// TIA Portal V17 export
// export: Created 2026-04-13T11:12:43.7188239Z, ExportSetting WithDefaults, DisplayName Totally Integrated Automation Portal, DisplayVersion V17 Update 4, DisplayName TIA Portal Openness, DisplayVersion V17 Update 4, DisplayName TIA Portal Version Control Interface, DisplayVersion V17, DisplayName SINAMICS Startdrive Advanced, DisplayVersion V17, DisplayName SINAMICS Startdrive G130, G150, S120, S150, SINAMICS MV, S210, DisplayVersion V17, DisplayName SINAMICS Startdrive G110M, G120, G120C, G120D, G120P, G115D, DisplayVersion V17, DisplayName STEP 7 Professional, DisplayVersion V17 Update 4, DisplayName STEP 7 Safety, DisplayVersion V17, DisplayName WinCC Professional, DisplayVersion V17 Update 4
FUNCTION_BLOCK "32-油炉控制"   // FB22, LAD
{ S7_Optimized_Access := 'FALSE' }
VERSION : 0.1
// stored: AutoNumber true, IsIECCheckEnabled false, SetENOAutomatically false, UDAEnableTagReadback false
   VAR_IN_OUT
      油炉温度写 : Real;
      油炉温度读 : Real;
      油炉循环泵启停 : Bool;
      油炉报警 : Bool;
      油炉冷却阀启停状态 : Bool;
      油炉加热泵启停状态 : Bool;
      油炉加热器1状态 : Bool;
      油炉加热器2状态 : Bool;
      油炉运行状态 : Bool;
      油炉自整定状态 : Bool;
      油炉强制冷却状态 : Bool;
      YL油炉温度写读 : Real;
   END_VAR
   VAR
      MB_COMM_LOAD { S7_SetPoint := 'True'} : Modbus_Comm_Load;
      MB_MASTER_DB { S7_SetPoint := 'True'} : Modbus_Master;
   END_VAR
   VAR DB_SPECIFIC
      CTU { S7_SetPoint := 'True'} : CTU_INT;
      TEMP { S7_SetPoint := 'True'} : Bool;
      TP : Array[0..40] of Bool;
      油炉温度读辅 : Int;
      油炉温度写辅 : Int;
      ST1 : Real;
      ST2 : Real;
      ST3 : Real;
      ST4 : Real;
      ST5 : Real;
      ST16 : Real;
      ST17 : Real;
      ST18 : Real;
      ST20 : Real;
      ST21 : Real;
      ST22 : Real;
      油炉状态1 : Int;
      油炉状态2 : Int;
      油炉启停字 : Int;
      油炉加热状态 : Int;
      油炉运行标志 : Int;
      YL油炉温度写读辅 : Int;
   END_VAR
   VAR
      Modbus_Comm_Load { S7_SetPoint := 'True'} : Modbus_Comm_Load;
      Modbus_Master { S7_SetPoint := 'True'} : Modbus_Master;
   END_VAR
   VAR_TEMP   // added for the SCL form of the ladder/FBD networks
      _w1 : Bool;
      _w2 : Bool;
      _w3 : Bool;
   END_VAR
BEGIN

REGION Network 1
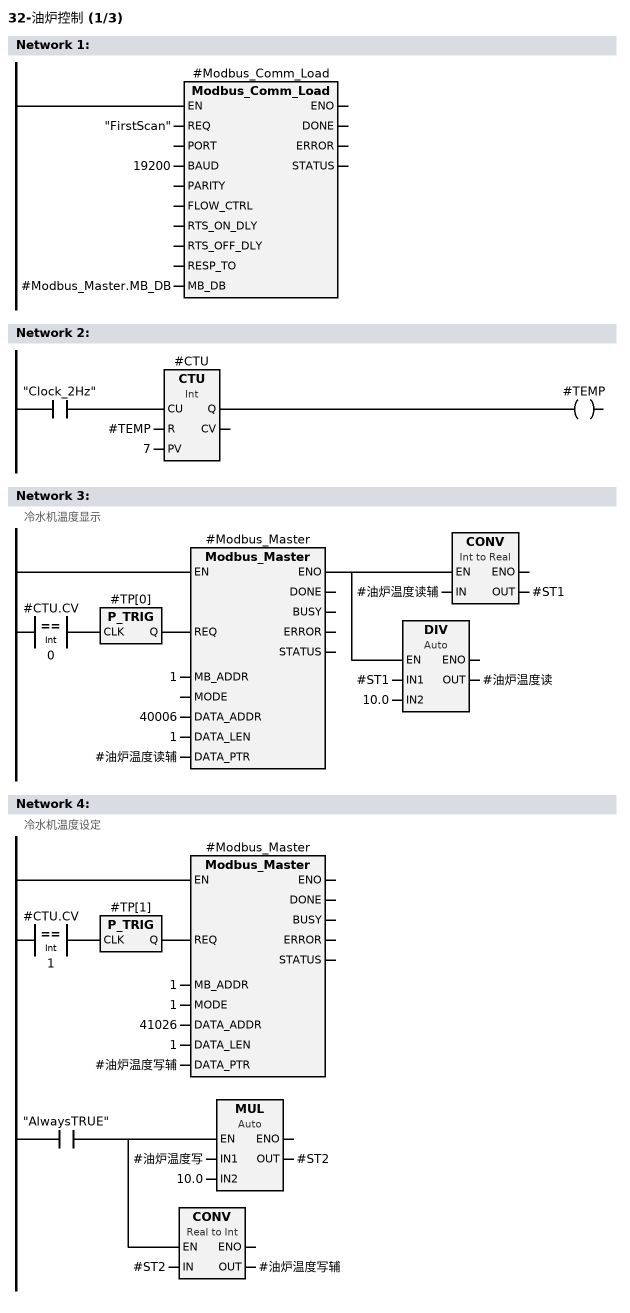
   RUNG wire#powerrail
      #Modbus_Comm_Load.Modbus_Comm_Load(REQ := "FirstScan", PORT :=, BAUD := 19200, PARITY :=, FLOW_CTRL :=, RTS_ON_DLY :=, RTS_OFF_DLY :=, RESP_TO :=, MB_DB := #Modbus_Master.MB_DB, DONE =>, ERROR =>, STATUS =>)
   END_RUNG
   // the same network as SCL:
   #Modbus_Comm_Load(REQ := "FirstScan", BAUD := 19200, MB_DB := #Modbus_Master.MB_DB);   // Modbus_Comm_Load
END_REGION

REGION Network 2
   RUNG wire#powerrail
      Contact( "Clock_2Hz" )
      { S7_Templates := "value_type := Int" } #CTU.CTU(r := #TEMP, pv := 7, cv =>)
      Coil( #TEMP )
   END_RUNG
   // the same network as SCL:
   #CTU(CU := "Clock_2Hz", R := #TEMP, PV := 7);   // CTU
   #TEMP := #CTU.Q;
END_REGION

REGION Network 3
   // 冷水机温度显示
   RUNG wire#powerrail
      #Modbus_Master.Modbus_Master(REQ := wire#w1, MB_ADDR := 1, MODE :=, DATA_ADDR := 40006, DATA_LEN := 1, DATA_PTR := #油炉温度读辅, DONE =>, BUSY =>, ERROR =>, STATUS =>)
      wire#w2
      { S7_Templates := "[SrcType := Int, DestType := Real]" } Convert(in := #油炉温度读辅, out => #ST1)
   END_RUNG
   RUNG wire#powerrail
      { S7_Templates := "SrcType := Int" } EQ_Contact(in1 := #CTU.CV, in2 := 0)
      P_Trig( #TP[0] )
   END_RUNG wire#w1
   RUNG wire#w2
      Div(in1 := #ST1, in2 := 10.0, out => #油炉温度读)
   END_RUNG
   // the same network as SCL:
   #_w1 := #CTU.CV = 0;
   #_w2 := #_w1 AND NOT #TP[0];   // rising edge
   #TP[0] := #_w1;
   #Modbus_Master(REQ := #_w2,   // Modbus_Master
                  MB_ADDR := 1,
                  DATA_ADDR := 40006,
                  DATA_LEN := 1,
                  DATA_PTR := #油炉温度读辅,
                  ENO => #_w3);
   IF #_w3 THEN
       #ST1 := INT_TO_REAL(#油炉温度读辅);
       #油炉温度读 := #ST1 / 10.0;
   END_IF;
END_REGION

REGION Network 4
   // 冷水机温度设定
   RUNG wire#powerrail
      #Modbus_Master.Modbus_Master(REQ := wire#w1, MB_ADDR := 1, MODE := 1, DATA_ADDR := 41026, DATA_LEN := 1, DATA_PTR := #油炉温度写辅, DONE =>, BUSY =>, ERROR =>, STATUS =>)
   END_RUNG
   RUNG wire#powerrail
      { S7_Templates := "SrcType := Int" } EQ_Contact(in1 := #CTU.CV, in2 := 1)
      P_Trig( #TP[1] )
   END_RUNG wire#w1
   RUNG wire#powerrail
      Contact( "AlwaysTRUE" )
      wire#w2
      Mul(in1 := #油炉温度写, in2 := 10.0, out => #ST2)
   END_RUNG
   RUNG wire#w2
      { S7_Templates := "[SrcType := Real, DestType := Int]" } Convert(in := #ST2, out => #油炉温度写辅)
   END_RUNG
   // the same network as SCL:
   #_w1 := #CTU.CV = 1;
   #_w2 := #_w1 AND NOT #TP[1];   // rising edge
   #TP[1] := #_w1;
   #Modbus_Master(REQ := #_w2, MB_ADDR := 1, MODE := 1, DATA_ADDR := 41026, DATA_LEN := 1, DATA_PTR := #油炉温度写辅);   // Modbus_Master
   IF "AlwaysTRUE" THEN
       #ST2 := #油炉温度写 * 10.0;
       #油炉温度写辅 := REAL_TO_INT(#ST2);
   END_IF;
END_REGION

REGION Network 5
   // 冷水机温度设定
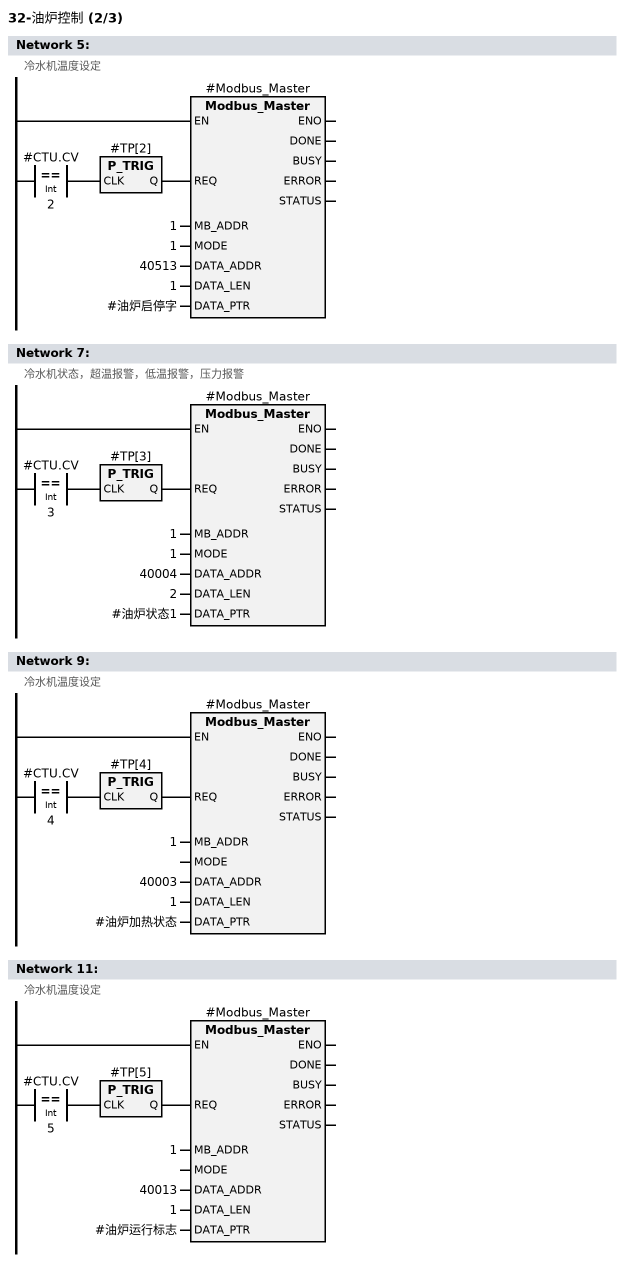
   RUNG wire#powerrail
      #Modbus_Master.Modbus_Master(REQ := wire#w1, MB_ADDR := 1, MODE := 1, DATA_ADDR := 40513, DATA_LEN := 1, DATA_PTR := #油炉启停字, DONE =>, BUSY =>, ERROR =>, STATUS =>)
   END_RUNG
   RUNG wire#powerrail
      { S7_Templates := "SrcType := Int" } EQ_Contact(in1 := #CTU.CV, in2 := 2)
      P_Trig( #TP[2] )
   END_RUNG wire#w1
   // the same network as SCL:
   #_w1 := #CTU.CV = 2;
   #_w2 := #_w1 AND NOT #TP[2];   // rising edge
   #TP[2] := #_w1;
   #Modbus_Master(REQ := #_w2, MB_ADDR := 1, MODE := 1, DATA_ADDR := 40513, DATA_LEN := 1, DATA_PTR := #油炉启停字);   // Modbus_Master
END_REGION

REGION Network 6 (SCL)
   IF #油炉循环泵启停 = TRUE THEN
       #油炉启停字:= 114;
   ELSE
       #油炉启停字 := 112;
   END_IF;
END_REGION

REGION Network 7
   // 冷水机状态，超温报警，低温报警，压力报警
   RUNG wire#powerrail
      #Modbus_Master.Modbus_Master(REQ := wire#w1, MB_ADDR := 1, MODE := 1, DATA_ADDR := 40004, DATA_LEN := 2, DATA_PTR := #油炉状态1, DONE =>, BUSY =>, ERROR =>, STATUS =>)
   END_RUNG
   RUNG wire#powerrail
      { S7_Templates := "SrcType := Int" } EQ_Contact(in1 := #CTU.CV, in2 := 3)
      P_Trig( #TP[3] )
   END_RUNG wire#w1
   // the same network as SCL:
   #_w1 := #CTU.CV = 3;
   #_w2 := #_w1 AND NOT #TP[3];   // rising edge
   #TP[3] := #_w1;
   #Modbus_Master(REQ := #_w2, MB_ADDR := 1, MODE := 1, DATA_ADDR := 40004, DATA_LEN := 2, DATA_PTR := #油炉状态1);   // Modbus_Master
END_REGION

REGION Network 8 (SCL)
   IF #油炉状态1>1 OR #油炉状态2>1 THEN
       #油炉报警 := TRUE;
   ELSE
       #油炉报警 := FALSE;
   END_IF;
END_REGION

REGION Network 9
   // 冷水机温度设定
   RUNG wire#powerrail
      #Modbus_Master.Modbus_Master(REQ := wire#w1, MB_ADDR := 1, MODE :=, DATA_ADDR := 40003, DATA_LEN := 1, DATA_PTR := #油炉加热状态, DONE =>, BUSY =>, ERROR =>, STATUS =>)
   END_RUNG
   RUNG wire#powerrail
      { S7_Templates := "SrcType := Int" } EQ_Contact(in1 := #CTU.CV, in2 := 4)
      P_Trig( #TP[4] )
   END_RUNG wire#w1
   // the same network as SCL:
   #_w1 := #CTU.CV = 4;
   #_w2 := #_w1 AND NOT #TP[4];   // rising edge
   #TP[4] := #_w1;
   #Modbus_Master(REQ := #_w2, MB_ADDR := 1, DATA_ADDR := 40003, DATA_LEN := 1, DATA_PTR := #油炉加热状态);   // Modbus_Master
END_REGION

REGION Network 10 (SCL)
   IF #油炉加热状态 >= 8 THEN
       #油炉冷却阀启停状态 := TRUE;
   ELSE
       #油炉冷却阀启停状态 := FALSE;
   END_IF;

   IF #油炉加热状态 >= 4 THEN
       #油炉加热泵启停状态 := TRUE;
   ELSE
       #油炉加热泵启停状态 := FALSE;
   END_IF;


   IF #油炉加热状态 >= 2 THEN
       #油炉加热器2状态 := TRUE;
   ELSE
       #油炉加热器2状态 := FALSE;
   END_IF;

   IF #油炉加热状态 >= 1 THEN
       #油炉加热器1状态 := TRUE;
   ELSE
       #油炉加热器1状态 := FALSE;
   END_IF;
END_REGION

REGION Network 11
   // 冷水机温度设定
   RUNG wire#powerrail
      #Modbus_Master.Modbus_Master(REQ := wire#w1, MB_ADDR := 1, MODE :=, DATA_ADDR := 40013, DATA_LEN := 1, DATA_PTR := #油炉运行标志, DONE =>, BUSY =>, ERROR =>, STATUS =>)
   END_RUNG
   RUNG wire#powerrail
      { S7_Templates := "SrcType := Int" } EQ_Contact(in1 := #CTU.CV, in2 := 5)
      P_Trig( #TP[5] )
   END_RUNG wire#w1
   // the same network as SCL:
   #_w1 := #CTU.CV = 5;
   #_w2 := #_w1 AND NOT #TP[5];   // rising edge
   #TP[5] := #_w1;
   #Modbus_Master(REQ := #_w2, MB_ADDR := 1, DATA_ADDR := 40013, DATA_LEN := 1, DATA_PTR := #油炉运行标志);   // Modbus_Master
END_REGION

REGION Network 12
   // 冷水机温du
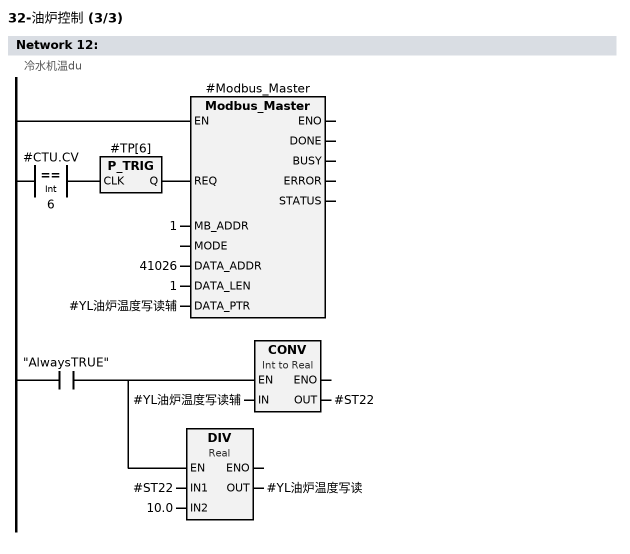
   RUNG wire#powerrail
      #Modbus_Master.Modbus_Master(REQ := wire#w1, MB_ADDR := 1, MODE :=, DATA_ADDR := 41026, DATA_LEN := 1, DATA_PTR := #YL油炉温度写读辅, DONE =>, BUSY =>, ERROR =>, STATUS =>)
   END_RUNG
   RUNG wire#powerrail
      { S7_Templates := "SrcType := Int" } EQ_Contact(in1 := #CTU.CV, in2 := 6)
      P_Trig( #TP[6] )
   END_RUNG wire#w1
   RUNG wire#powerrail
      Contact( "AlwaysTRUE" )
      wire#w2
      { S7_Templates := "[SrcType := Int, DestType := Real]" } Convert(in := #YL油炉温度写读辅, out => #ST22)
   END_RUNG
   RUNG wire#w2
      { S7_Templates := "SrcType := Real" } Div(in1 := #ST22, in2 := 10.0, out => #YL油炉温度写读)
   END_RUNG
   // the same network as SCL:
   #_w1 := #CTU.CV = 6;
   #_w2 := #_w1 AND NOT #TP[6];   // rising edge
   #TP[6] := #_w1;
   #Modbus_Master(REQ := #_w2, MB_ADDR := 1, DATA_ADDR := 41026, DATA_LEN := 1, DATA_PTR := #YL油炉温度写读辅);   // Modbus_Master
   IF "AlwaysTRUE" THEN
       #ST22 := INT_TO_REAL(#YL油炉温度写读辅);
       #YL油炉温度写读 := #ST22 / 10.0;
   END_IF;
END_REGION

REGION Network 13 (SCL)
   IF #油炉运行标志 >= 4 THEN
       #油炉强制冷却状态 := TRUE;
   ELSE
       #油炉强制冷却状态 := FALSE;
   END_IF;

   IF #油炉运行标志 >= 2 THEN
       #油炉自整定状态 := TRUE;
   ELSE
       #油炉自整定状态 := FALSE;
   END_IF;


   IF #油炉运行标志 >= 1 THEN
       #油炉运行状态 := TRUE;
   ELSE
       #油炉运行状态 := FALSE;
   END_IF;
END_REGION
END_FUNCTION_BLOCK
